FUNCTION FC_8strConcatSeparator : T_DEFAULT_STR
VAR_INPUT
	iSeparator:		STRING := IING.STRING_UNDERSCORE;
	iStr1:			T_DEFAULT_STR;
	iStr2:			T_DEFAULT_STR;
	iStr3:			T_DEFAULT_STR;
	iStr4:			T_DEFAULT_STR;
	iStr5:			T_DEFAULT_STR;
	iStr6:			T_DEFAULT_STR;
	iStr7:			T_DEFAULT_STR;
	iStr8:			T_DEFAULT_STR;
END_VAR

FC_8strConcatSeparator := FC_2strConcatSeparator(iSeparator, FC_7strConcatSeparator(iSeparator, iStr1, iStr2, iStr3, iStr4, iStr5, iStr6, iStr7), iStr8);

END_FUNCTION

(* stored: Version 1.1.0.1, ProductVersion 3.1.4026.18
   POU FC_8strConcatSeparator: Id {ce126934-3bf9-45bd-b4cb-e3c6390a01a6}, SpecialFunc None *)
